// TIA Portal V20 export
FUNCTION "LBP_CallBackAuxFunc" : Void   // FC12, SCL
TITLE = Auxiliary functions / Fonctions auxiliaires
{ S7_Optimized_Access := 'FALSE' }
AUTHOR : SINUMERIK
FAMILY : SINUMERIK_ONE
VERSION : 6.24
// Call interface for users for auxiliary functions, the block is called on an event-driven basis in the basic program when new auxiliary functions are available / Interface d'appel pour utilisateurs de fonctions auxiliaires. Le bloc est appelé dans le programme de base sur événement lorsque de nouvelles fonctions auxiliaires sont disponibles
// stored: AutoNumber false, IsIECCheckEnabled true, SetENOAutomatically false
   VAR_INPUT
      Chan : Byte;   // Index of channel / Indice de canal
   END_VAR
BEGIN
END_FUNCTION
